FUNCTION_BLOCK OPTIMIZE_MODELS
  {SET_ATTRIBUTE(OpcUa, SERVICE)}
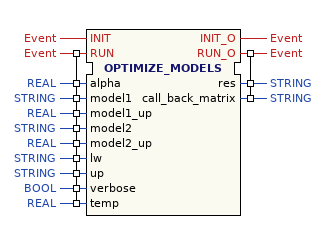
  EVENT_INPUT
    INIT;
    RUN WITH alpha, model1, model1_up, model2, model2_up, lw, up, verbose, temp; {SET_ATTRIBUTE(OpcUa, Method)}
  END_EVENT
  EVENT_OUTPUT
    INIT_O;
    RUN_O WITH res, call_back_matrix;
  END_EVENT
  VAR_INPUT
    alpha : REAL; {SET_ATTRIBUTE(OpcUa, Variable.RUN)}
    model1 : STRING; {SET_ATTRIBUTE(OpcUa, Variable.RUN)}
    model1_up : REAL; {SET_ATTRIBUTE(OpcUa, Variable.RUN)}
    model2 : STRING; {SET_ATTRIBUTE(OpcUa, Variable.RUN)}
    model2_up : REAL; {SET_ATTRIBUTE(OpcUa, Variable.RUN)}
    lw : STRING; {SET_ATTRIBUTE(OpcUa, Variable.RUN)}
    up : STRING; {SET_ATTRIBUTE(OpcUa, Variable.RUN)}
    verbose : BOOL; {SET_ATTRIBUTE(OpcUa, Variable.RUN)}
    temp : REAL; {SET_ATTRIBUTE(OpcUa, Variable.RUN)}
  END_VAR
  VAR_OUTPUT
    res : STRING; {SET_ATTRIBUTE(OpcUa, Variable.RUN)}
    call_back_matrix : STRING; {SET_ATTRIBUTE(OpcUa, Variable.RUN)}
  END_VAR
END_FUNCTION_BLOCK
